// TwinCAT 3 PLC project SmartHomeDevices_ReferenceLibrary
// Title: Smart Home Device Library
// Company: Oleksandr Tiutyk
// ProjectVersion: 0.0.0.1
// Description: OOP conceps demo for smart home
// ProgramVersion: 3.1.4026.20
// libraries:
//   [Smart Home Library], * (Oleksandr Tiutyk)
//   Tc2_Standard, * (Beckhoff Automation GmbH)
//   Tc2_System, * (Beckhoff Automation GmbH)
// project tree:
//   InputDevices/ CarbonDioxideSensor.TcPOU
//   InputOutputDevices/ ClimatSystem.TcPOU
//   / Device.TcPOU
//   OutputDevices/ Ventilation.TcPOU
// (motion and I/O tree: see PLC project smarthome_referencelibrary)
// real-time tasks:
//   TASK PlcTask: cycle T#10ms, priority 20, ADS port 350
//   TASK PlcTask1: cycle T#10ms, priority 21, ADS port 351

// ---- InputDevices/CarbonDioxideSensor.TcPOU
FUNCTION_BLOCK CarbonDioxideSensor EXTENDS Device IMPLEMENTS SHLib.IInputDevice
VAR
	_CarbonDioxideLevel : WORD := 800;
	
	_MappedValue AT %Q* : WORD;
END_VAR

{attribute 'monitoring' := 'call'}
PROPERTY CarbonDioxideLevel : WORD
GET
CarbonDioxideLevel := _CarbonDioxideLevel;
END_GET
END_PROPERTY

{attribute 'monitoring' := 'call'}
PROPERTY Name : STRING
GET
Name := 'CarbonDioxideSensor';
END_GET
END_PROPERTY

METHOD ReadInputs
// handle value from terminal here
END_METHOD

END_FUNCTION_BLOCK

// ---- Device.TcPOU
FUNCTION_BLOCK ABSTRACT Device IMPLEMENTS SHLib.IDevice
VAR_INPUT
	ErrorSimulation : BOOL;
END_VAR
VAR
	_Place : STRING;
END_VAR

//FB_Init is always available implicitly and it is used primarily for initialization.
//The return value is not evaluated. For a specific influence, you can also declare the
//methods explicitly and provide additional code there with the standard initialization
//code. You can evaluate the return value.
METHOD FB_Init: BOOL
VAR_INPUT
    bInitRetains: BOOL; // TRUE: the retain variables are initialized (reset warm / reset cold)
    bInCopyCode: BOOL;  // TRUE: the instance will be copied to the copy code afterward (online change)   
	place : STRING;
END_VAR
_Place := place;
END_METHOD

{attribute 'monitoring' := 'call'}
PROPERTY ABSTRACT Name : STRING
GET
END_GET
END_PROPERTY

{attribute 'monitoring' := 'call'}
PROPERTY FINAL Place : STRING
GET
Place := _Place;
END_GET
END_PROPERTY

{attribute 'monitoring' := 'call'}
PROPERTY FINAL State : SHLib.DEVICE_STATE
GET
IF ErrorSimulation THEN
	State := SHLib.DEVICE_STATE.FAULT;
ELSE
	State := SHLib.DEVICE_STATE.WORKING;
END_IF
END_GET
END_PROPERTY

END_FUNCTION_BLOCK

// ---- InputOutputDevices/ClimatSystem.TcPOU
FUNCTION_BLOCK ClimatSystem EXTENDS Device IMPLEMENTS SHLib.IInputDevice, SHLib.IOutputDevice
VAR
	_Temperature : SINT := 25;
	
	_IsCoolingOn : BOOL;
	_IsHeatingOn : BOOL;
END_VAR

{attribute 'monitoring' := 'call'}
PROPERTY IsCoolingOn : BOOL
GET
IsCoolingOn := _IsCoolingOn;
END_GET
END_PROPERTY

{attribute 'monitoring' := 'call'}
PROPERTY IsHeatingOn : BOOL
GET
IsHeatingOn := _IsHeatingOn;
END_GET
END_PROPERTY

{attribute 'monitoring' := 'call'}
PROPERTY Name : STRING
GET
Name := 'ClimatSystem';
END_GET
END_PROPERTY

METHOD ReadInputs
// handle value from terminal here
END_METHOD

{attribute 'monitoring' := 'call'}
PROPERTY Temperature : SINT
GET
Temperature := _Temperature;
END_GET
END_PROPERTY

METHOD WriteOutputs
_IsHeatingOn := _Temperature <= 20;
_IsCoolingOn := _Temperature >= 30;
END_METHOD

END_FUNCTION_BLOCK

// ---- OutputDevices/Ventilation.TcPOU
FUNCTION_BLOCK Ventilation EXTENDS Device IMPLEMENTS SHLib.IOutputDevice
VAR
	_Speed : BYTE;
END_VAR

{attribute 'monitoring' := 'call'}
PROPERTY IsOn : BOOL
GET
IsOn := _Speed <> 0;
END_GET
END_PROPERTY

{attribute 'monitoring' := 'call'}
PROPERTY Name : STRING
GET
Name := 'Ventilation';
END_GET
END_PROPERTY

METHOD SetSpeed
VAR_INPUT
	speed : BYTE;
END_VAR
_Speed := speed;
END_METHOD

{attribute 'monitoring' := 'call'}
PROPERTY Speed : BYTE
GET
Speed := _Speed;
END_GET
END_PROPERTY

METHOD WriteOutputs
// put values to terminal here
END_METHOD

END_FUNCTION_BLOCK
